{attribute 'linkalways'} 
{attribute 'no_explicit_call' := 'This FB is a CLASS and must be accessed using methods or properties'}
{attribute 'enable_dynamic_creation'}
FUNCTION_BLOCK _ETcVnSvm EXTENDS EnumDatatypeBase
VAR
	localData : ETcVnSvm;
	activeData : REFERENCE TO ETcVnSvm;
	enumBaseDatatype : _UDINT(localData);
END_VAR

METHOD PRIVATE AddLocalEnumeration
VAR_INPUT
	Enumeration : T_MAXSTRING;
	Value : ETcVnSvm;
END_VAR
AddEnumeration(Enumeration, Value);
END_METHOD

PROPERTY PUBLIC Address : PVOID
GET
Address := ADR(activeData);
END_GET
END_PROPERTY

METHOD PUBLIC ClearReference
VAR_INPUT
END_VAR
activeData REF= localData;
SetBaseDatatypeReference();
END_METHOD

METHOD PUBLIC Clone : I_Datatype
VAR
    pClone : POINTER TO _ETcVnSvm;
END_VAR
pClone := __NEW(_ETcVnSvm(InitialValue := Value));
Clone := pClone^;
END_METHOD

METHOD FB_init : BOOL
VAR_INPUT
	bInitRetains : BOOL; // if TRUE, the retain variables are initialized (warm start / cold start)
	bInCopyCode : BOOL;  // if TRUE, the instance afterwards gets moved into the copy code (online change)
	InitialValue : ETcVnSvm;
END_VAR
localData := InitialValue;
AddBaseDatatype(enumBaseDatatype);
ClearReference();

AddLocalEnumeration('TCVN_SVM_C_CLASSIFIER', ETcVnSvm.TCVN_SVM_C_CLASSIFIER);
AddLocalEnumeration('TCVN_SVM_NU_CLASSIFIER', ETcVnSvm.TCVN_SVM_NU_CLASSIFIER);
AddLocalEnumeration('TCVN_SVM_NOVELTY_DETECTOR', ETcVnSvm.TCVN_SVM_NOVELTY_DETECTOR);
AddLocalEnumeration('TCVN_SVM_EPS_REGRESSOR', ETcVnSvm.TCVN_SVM_EPS_REGRESSOR);
AddLocalEnumeration('TCVN_SVM_NU_REGRESSOR', ETcVnSvm.TCVN_SVM_NU_REGRESSOR);
END_METHOD

PROPERTY PUBLIC Identifier : T_MAXSTRING
GET
Identifier := 'ETcVnSvm';
END_GET
END_PROPERTY

METHOD IsEnumeratorValueEqual : BOOL
VAR_INPUT
	Enumerator : I_KeyValueForwardEnumerator;
END_VAR
VAR
	storedValue : ETcVnSvm;
END_VAR
IF NOT Enumerator.TryGet(storedValue) THEN
	RETURN;
END_IF

IsEnumeratorValueEqual := storedValue = activeData;
END_METHOD

METHOD PUBLIC MakeReferenceTo
VAR_INPUT
	ReferenceTarget : REFERENCE TO ETcVnSvm;
END_VAR
activeData REF= ReferenceTarget;
SetBaseDatatypeReference();
END_METHOD

METHOD PROTECTED SetBaseDatatypeReference
VAR_INPUT
END_VAR
enumBaseDatatype.MakeReferenceTo(activeData);
END_METHOD

PROPERTY PUBLIC Size : UDINT
GET
Size := SIZEOF(activeData);
END_GET
END_PROPERTY

METHOD TryMakeReferenceTo : BOOL
VAR_INPUT
	Target : I_Datatype;
END_VAR
VAR
	targetAsEnum : I_EnumDatatype;
	pTargetData : POINTER TO ETcVnSvm;
END_VAR
IF NOT Target.TryResolveAsEnumDatatype(targetAsEnum) THEN
	RETURN;
END_IF

IF targetAsEnum.Identifier <> Identifier THEN
	RETURN;
END_IF

pTargetData := Target.Address;
activeData REF= pTargetData^;
SetBaseDatatypeReference();
TryMakeReferenceTo := TRUE;
END_METHOD

PROPERTY PUBLIC Value : ETcVnSvm
GET
Value := activeData;
END_GET
SET
activeData := Value;
END_SET
END_PROPERTY

END_FUNCTION_BLOCK

(* stored: Version 1.1.0.1
   POU _ETcVnSvm: Id {bb1946a4-4401-4f72-a4d8-271c6b73eda5}, SpecialFunc None
   Folder Constructor: Id {d7407a7c-4174-4135-8335-11233af70b84}
   Folder Private: Id {4a666c42-c0e7-48cb-83f5-fdd1d5559008}
   Folder Protected: Id {282e832f-431d-4845-ab5f-635a2a2d84e5}
   Method AddLocalEnumeration: Id {376a6c07-e997-437e-8efc-6f4c3dfb1f10}
   Property Address: Id {6676b53e-f89f-44ce-b188-97466a95beb6}
   Get Get: Id {8360599c-74d7-4b13-98b4-9eba997b42ae}
   Method ClearReference: Id {d5342cc7-ca6f-4196-b149-229caeb810ec}
   Method Clone: Id {2bcd65d1-1cbe-418b-8d17-7e2752b169bd}
   Method FB_init: Id {77183120-d9a1-44ae-8fbf-ecd9484748e1}
   Property Identifier: Id {83a6a1c0-618a-4697-a0d5-d5918f04eb35}
   Get Get: Id {8eb1cefc-7580-4da7-b359-7bcc3ba00527}
   Method IsEnumeratorValueEqual: Id {8356a2f5-6669-4e3d-baf2-b62aaf4b307f}
   Method MakeReferenceTo: Id {b2f5f19e-7710-45b0-9853-c90b43331206}
   Method SetBaseDatatypeReference: Id {fa651099-b73d-49b5-b629-2948aeef85f9}
   Property Size: Id {85fb2d3c-c6f5-4623-b102-fef1cf1f8716}
   Get Get: Id {b3b60819-7a24-429a-867c-8647cf543dcc}
   Method TryMakeReferenceTo: Id {60eda7f7-a9ce-4e0e-a50f-15f9a26a9489}
   Property Value: Id {64a24fab-3b07-4d29-b3c6-b65dff98d5f5}
   Get Get: Id {e34e977d-6aec-4c70-98c3-e6ea8f1ec570}
   Set Set: Id {5a941163-c023-4858-9dbb-a198014a9223} *)
